// TIA Portal V20 export
VAR_GLOBAL   // PLC tag table "LKinCtrl_Configuration"
END_VAR
VAR_GLOBAL CONSTANT   // user constants
   LKINCTRL_SPTP_EXECUTION_STATUS_OUTPUT : Int := 0;   // 0: Regular time status; 1: Inverted time status; 2: Approximate cartesian distance
   LKINCTRL_LENGTH_OF_OFFSET_NAME : Int := 20;   // length of offset name / Length of offset name
   LKINCTRL_DISABLE_FLAG_RESET : Bool := TRUE;   // FALSE: Reset with execute & after done ; TRUE: No reset
   LKINCTRL_NO_OF_OFFSETS : Int := 3;   // number of configurable offsets / Number of configurable offsets
   LKINCTRL_NO_OF_START_EXECUTE_CMDS : Int := 1;   // number of cmds to be buffered in first cycle / Number of cmds to be buffered in first cycle
   LKINCTRL_LENGTH_OF_CMDPOINT_NAME : Int := 30;   // length of point name / Length of point name
   LKINCTRL_NO_OF_CONVEYOR : Int := 5;   // number of configurable offsets / Number of configurable offsets
   LKINCTRL_NO_OF_SEQ_EXECUTE_CMDS : Int := 1;   // number of cmds to be buffered after first cycle / Number of cmds to be buffered after first cycle
   LKINCTRL_NO_OF_CMD_VALUEFLAGS : Int := 4;   // number of LREAL flags per command / Number of LREAL flags per command
   LKINCTRL_NO_OF_ZONES : Int := 10;   // number of zone definitions / Number of zone definitions
   LKINCTRL_NO_OF_PATHDATA_ELEMENTS : Int := 20;   // length of LKinCtrl_typePathData / Length of LKinCtrl_typePathData
   LKINCTRL_NO_OF_CMD_SETFLAGS : Int := 3;   // number of Boolean flags per command / Number of Boolean flags per command
   LKINCTRL_LENGTH_OF_PATHDATA_NAME : Int := 20;   // length of PathData name / Length of PathData name
   LKINCTRL_NO_OF_POINTS_AT_POINT_TABLE : Int := 30;   // Number of points at point table. Valid values are 1..x
   LKINCTRL_LENGTH_OF_TO_NAME : UInt := 30;   // Maximum number of characters for technology object name.
   LKINCTRL_NO_OF_LAST_VALUEFLAG : Int := 30;   // Number of value flags at MovePath FB
   LKINCTRL_NO_OF_LAST_SETFLAG : Int := 30;   // Number of flags at MovePath FB
   LKINCTRL_NO_OF_PATHS : Int := 5;   // Number of paths. Valid values are 1..x
END_VAR
